FUNCTION_BLOCK FB_WritePWM
VAR_INPUT
	bExecute : BOOL := FALSE;
	slv_addr : UINT := 0;
	value : REAL := 0.0;
END_VAR
VAR_OUTPUT
	state : INT := 0;
	bError : BOOL;
END_VAR
VAR
	fbSdoWrite : FB_EcCoESdoWrite;
	nErrID : UDINT :=0;
	sdo_address: UINT := 16#8001;
	subIndex: BYTE := 7;
END_VAR

fbSdoWrite(
        sNetId          := MAIN.sNetId_local,
        //nSlaveAddr      := nSlaveAddr,
		nSlaveAddr :=   slv_addr,
        nIndex          := sdo_address,
        nSubIndex       := subIndex,
        pSrcBuf         := ADR(value),
        cbBufLen        := SIZEOF(value),
        bExecute        := bExecute
);
state := 1;
IF NOT fbSdoWrite.bBusy THEN
        bExecute := FALSE;
		//done	:= TRUE;
        IF NOT fbSdoWrite.bError THEN 
                (* write successful *)
                bError := FALSE;
                nErrId := 0;
        ELSE 
                (* write failed *)
                bError := fbSdoWrite.bError;
                nErrId := fbSdoWrite.nErrId;
        END_IF
        fbSdoWrite(bExecute := FALSE);
		state := 0;
END_IF

END_FUNCTION_BLOCK

(* stored: Version 1.1.0.1, ProductVersion 3.1.4024.10
   POU FB_WritePWM: Id {c1b9dc75-7f30-47d3-9658-10e6396613d9}, SpecialFunc None *)
